INTERFACE I_CoE_property_handler

METHOD add_read_request : BOOL
VAR_INPUT
	request	: I_CoE_property;
END_VAR
END_METHOD

METHOD add_write_request : BOOL
VAR_INPUT
	request	: I_CoE_property;
END_VAR
END_METHOD

END_INTERFACE

(* stored: Version 1.1.0.1, ProductVersion 3.1.4024.6
   Itf I_CoE_property_handler: Id {b4af1cd9-bdfe-0ee1-2d64-f13c9b6da31f}
   Method add_read_request: Id {4b6a293e-3229-075a-2c2a-594477e299fa}
   Method add_write_request: Id {15246adc-202f-07b7-038d-9188c1207b35} *)
